// TIA Portal V15 export
// export: Created 2018-05-29T12:25:38.1552518Z, ExportSetting WithDefaults, DisplayName Totally Integrated Automation Portal, DisplayVersion V15, DisplayName STEP 7 Professional, DisplayVersion V15, DisplayName WinCC Professional, DisplayVersion V15, DisplayName TIA Portal Openness, DisplayVersion V15
FUNCTION "T109_fc" : Void   // FC1, STL
TITLE = _fc
{ S7_Optimized_Access := 'TRUE' }
VERSION : 0.1
// test
// stored: AutoNumber true, UDAEnableTagReadback false
BEGIN

NETWORK
TITLE = Main


// code


END_FUNCTION
